  MoveL 720 to (339.04, 119.32, 0) mm, rotated rx 180 ry 0 rz 119.57 deg; joints [20.503, -55.364, 119.544, -42.913, -70.488, 17.251]
  MoveL 721 to (338.35, 118.95, 0) mm, rotated rx -180 ry 0 rz 119.57 deg; joints [20.529, -55.385, 119.588, -42.882, -70.496, 17.226]
  MoveL 722 to (337.63, 118.65, 0) mm, rotated rx 180 ry 0 rz 119.57 deg; joints [20.552, -55.409, 119.635, -42.853, -70.507, 17.202]
  MoveL 723 to (336.88, 118.42, 0) mm, rotated rx 180 ry 0 rz 119.57 deg; joints [20.573, -55.435, 119.686, -42.826, -70.519, 17.176]
  MoveL 724 to (336.12, 118.25, 0) mm, rotated rx -180 ry 0 rz 119.57 deg; joints [20.591, -55.462, 119.741, -42.8, -70.534, 17.15]
  MoveL 725 to (335.34, 118.14, 0) mm, rotated rx -180 ry 0 rz 119.57 deg; joints [20.607, -55.491, 119.799, -42.777, -70.55, 17.124]
  MoveL 726 to (334.56, 118.11, 0) mm, rotated rx -180 ry 0 rz 119.57 deg; joints [20.621, -55.522, 119.859, -42.756, -70.568, 17.098]
  MoveL 727 to (320.08, 118.11, 0) mm, rotated rx -180 ry 0 rz 119.57 deg; joints [20.845, -56.086, 120.981, -42.397, -70.914, 16.623]
  MoveL 728 to (319.04, 118.17, 0) mm, rotated rx 180 ry 0 rz 119.57 deg; joints [20.859, -56.127, 121.064, -42.374, -70.941, 16.589]
  MoveL 729 to (318.02, 118.35, 0) mm, rotated rx 180 ry 0 rz 119.57 deg; joints [20.867, -56.169, 121.148, -42.355, -70.969, 16.556]
  MoveL 730 to (317.03, 118.65, 0) mm, rotated rx 180 ry 0 rz 119.57 deg; joints [20.871, -56.212, 121.233, -42.342, -70.999, 16.525]
  MoveL 731 to (316.08, 119.06, 0) mm, rotated rx 180 ry 0 rz 119.57 deg; joints [20.869, -56.255, 121.318, -42.334, -71.031, 16.495]
  MoveL 732 to (315.18, 119.58, 0) mm, rotated rx -180 ry 0 rz 119.57 deg; joints [20.861, -56.297, 121.402, -42.332, -71.064, 16.468]
  MoveL 733 to (314.36, 120.21, 0) mm, rotated rx 180 ry 0 rz 119.57 deg; joints [20.848, -56.338, 121.484, -42.336, -71.098, 16.444]
  MoveL 734 to (313.63, 120.94, 0) mm, rotated rx 180 ry 0 rz 119.57 deg; joints [20.829, -56.378, 121.562, -42.346, -71.132, 16.422]
  MoveL 735 to (312.99, 121.78, 0) mm, rotated rx -180 ry 0 rz 119.57 deg; joints [20.805, -56.415, 121.636, -42.362, -71.166, 16.404]
  MoveL 736 to (282.68, 167.64, 0) mm, rotated rx -180 ry 0 rz 119.57 deg; joints [19.335, -58.227, 125.238, -43.453, -72.882, 15.581]
  MoveL 737 to (268.12, 167.64, 0) mm, rotated rx -180 ry 0 rz 119.57 deg; joints [19.558, -58.782, 126.342, -43.113, -73.222, 15.123]
  MoveL 738 to (278.19, 152.4, 0) mm, rotated rx -180 ry 0 rz 119.57 deg; joints [20.061, -58.19, 125.164, -42.728, -72.662, 15.391]
  MoveL 739 to (288.26, 137.16, 0) mm, rotated rx -180 ry 0 rz 119.57 deg; joints [20.552, -57.589, 123.972, -42.359, -72.094, 15.66]
  MoveL 740 to (298.33, 121.92, 0) mm, rotated rx -180 ry 0 rz 119.57 deg; joints [21.032, -56.982, 122.763, -42.005, -71.518, 15.933]
  Set speed (2000.0 mm/s)
  MoveL 741 to (298.33, 121.92, 0) mm, rotated rx -180 ry 0 rz 119.57 deg; joints [21.032, -56.982, 122.763, -42.005, -71.518, 15.933]
  MoveL 742 to (298.33, 121.92, 10) mm, rotated rx -180 ry 0 rz 119.57 deg; joints [21.032, -57.583, 122.737, -42.148, -71.052, 16.377]
